ABB RobotStudio station: Project2.rsstnx

Station Project2 (saved by RobotStudio 25.2.11266.1)
Controller IRB120_3_58
  mechanical unit ROB_1: IRB120_3_58__01, 6 joints, base frame (0, 0, 0) mm
Layout (positions relative to the parent item):
  - IRB120_3_58__01 [mechanism, from %ABB.RobotStudio.Models.IRB120%\IRB120_3_58_G_01.rslib] at (0, 0, 0) mm; joint values [0.8069, 0.1269, -0.2176, -0.0228, 1.4767, 1.2827] (rad or m)
  - tool [part] at (-380.53, 565.66, 550.87) mm, rotated rx 16.99 ry 54.5 rz -12.92 deg, size 142.4 x 50 x 96.7 mm
  - Group_1 [graphiccomponentgroup]
  - work_object [part], size 424.3 x 424.3 x 300 mm
Attachment: tool is attached to IRB120_3_58__01 / Link6
Targets, tools, work objects and paths stored in the station, written as RAPID:
! task T_ROB1
MODULE CalibData
  TASK PERS wobjdata box:=[FALSE,TRUE,"",[[299.719,150.281,300],[0,0.382683432,0.923879533,0]],[[0,0,0],[1,0,0,0]]];
ENDMODULE

